Universal Robots PolyScope program: tarea_comandos.urp

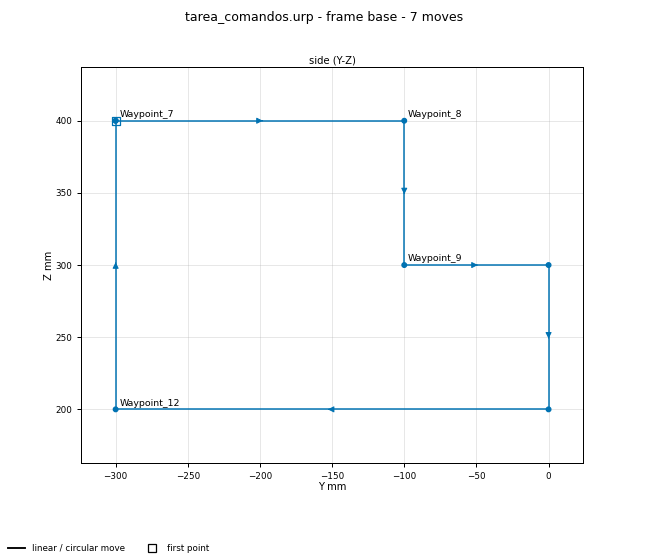
[picture p0: tool path of tarea_comandos.urp in frame base, 7 of 14 moves have a stored position in this frame; points joined in program order, loops and branches not executed]
Program tarea_comandos (installation=default directory=/home/hugo/Documents/Proyecto_Ingenieria/ursim-5.10.2.106319/programs/ASM/Clase1_Comandos createdIn=5.10.2.106319 lastSavedIn=5.10.2.106319 robotSerialNumber=20195599999)
Calibrated DH parameters: a=[0, -0.425, -0.3922, 0, 0, 0]; d=[0.1625, 0, 0, 0.1333, 0.0997, 0.0996]; alpha=[1.570796, 0, 0, 1.570796, -1.570796, 0]; deltaTheta=[0, 0, 0, 0, 0, 0]
Robot Program (runOnlyOnce=false)
  movimiento :=  (valueSource=Operator message=Elige Movimiento [1 - Relativos, 2 - Absolutos, 3 - Problema] valueType=Integer)
  repeticiones :=  (valueSource=Operator message=Introduce cantidad de repeticiones valueType=Integer)
  Loop While (checkContinuously=false) expression=repeticiones
    Switch expression=movimiento
      Case (caseValue=1)
        Folder Movimiento 1
          MoveL speed 250 mm/s, acceleration 1200 mm/s^2 (useActiveTCP=true) feature=Base
            Waypoint Waypoint_1 (Relative): relativeFromPosition TCP in base x=200 y=-300 z=400 mm, rx=-0.0013 ry=3.1193 rz=0.0359 rad; joints [-35.148, -69.126, -119.753, -80.848, 91.806, 54.808] deg; TCP in base x=200 y=-300 z=400 mm, rx=-0.0013 ry=3.1193 rz=0.0359 rad; joints [-35.148, -69.126, -119.753, -80.848, 91.806, 54.808] deg
            Waypoint Waypoint_2 (Relative): relativeFromPosition TCP in base x=200 y=-300 z=400 mm, rx=-0.0012 ry=3.1163 rz=0.0389 rad; joints [-35.205, -69.129, -119.772, -80.75, 91.997, 54.757] deg; TCP in base x=200 y=-100 z=400 mm, rx=-0.0012 ry=3.1163 rz=0.0389 rad; joints [9.378, -42.937, -130.525, -94.888, 91.177, 99.35] deg
            Waypoint Waypoint_3 (Relative): relativeFromPosition TCP in base x=200 y=-100 z=400 mm, rx=-0.0012 ry=3.1163 rz=0.0389 rad; joints [9.378, -42.937, -130.525, -94.888, 91.177, 99.35] deg; TCP in base x=200 y=-100 z=300 mm, rx=-0.0012 ry=3.1163 rz=0.0389 rad; joints [9.378, -43.258, -145.11, -79.982, 91.177, 99.35] deg
            Waypoint Waypoint_4 (Relative): relativeFromPosition TCP in base x=200 y=-100 z=300 mm, rx=-0.0012 ry=3.1163 rz=0.0389 rad; joints [9.378, -43.258, -145.11, -79.982, 91.177, 99.35] deg; TCP in base x=200 y=0 z=300 mm, rx=-0.0012 ry=3.1163 rz=0.0389 rad; joints [41.723, -35.535, -146.437, -86.004, 90.112, 131.68] deg
            Waypoint Waypoint_5 (Relative): relativeFromPosition TCP in base x=200 y=0 z=300 mm, rx=-0.0012 ry=3.1163 rz=0.0389 rad; joints [41.723, -35.535, -146.437, -86.004, 90.112, 131.68] deg; TCP in base x=200 y=0 z=200 mm, rx=-0.0012 ry=3.1163 rz=0.0389 rad; joints [41.723, -41.975, -160.626, -65.375, 90.112, 131.68] deg
            Waypoint Waypoint_6 (Relative): relativeFromPosition TCP in base x=200 y=0 z=200 mm, rx=-0.0012 ry=3.1163 rz=0.0389 rad; joints [41.723, -41.975, -160.626, -65.375, 90.112, 131.68] deg; TCP in base x=200 y=-300 z=200 mm, rx=-0.0012 ry=3.1163 rz=0.0389 rad; joints [-35.205, -85.851, -141.282, -42.519, 91.997, 54.757] deg
            Waypoint Waypoint_13 (Relative): relativeFromPosition TCP in base x=200 y=-300 z=200 mm, rx=-0.0012 ry=3.1163 rz=0.0389 rad; joints [-35.205, -85.851, -141.282, -42.519, 91.997, 54.757] deg; TCP in base x=200 y=-300 z=400 mm, rx=-0.0012 ry=3.1163 rz=0.0389 rad; joints [-35.205, -69.129, -119.772, -80.75, 91.997, 54.757] deg
      Case (caseValue=2)
        Folder Movimiento 2
          MoveL speed 250 mm/s, acceleration 1200 mm/s^2 (useActiveTCP=true) feature=Base
            Waypoint Waypoint_7: TCP in base x=200 y=-300 z=400 mm, rx=-0.0013 ry=3.1195 rz=0.0358 rad; joints [-35.145, -69.126, -119.751, -80.853, 91.797, 54.811] deg
            Waypoint Waypoint_8: motionParameters(blendRadius=0.05); TCP in base x=200 y=-100 z=400 mm, rx=-0.0013 ry=3.1195 rz=0.0358 rad; joints [9.426, -42.984, -130.463, -95.1, 91.091, 99.391] deg
            Waypoint Waypoint_9: motionParameters(blendRadius=0.05); TCP in base x=200 y=-100 z=300 mm, rx=-0.0013 ry=3.1195 rz=0.0358 rad; joints [9.426, -43.298, -145.05, -80.2, 91.091, 99.391] deg
            Waypoint Waypoint_10: motionParameters(blendRadius=0.05); TCP in base x=200 y=0 z=300 mm, rx=-0.0013 ry=3.1195 rz=0.0358 rad; joints [41.7, -35.632, -146.369, -86.188, 90.147, 131.654] deg
            Waypoint Waypoint_11: TCP in base x=200 y=0 z=200 mm, rx=-0.0013 ry=3.1195 rz=0.0358 rad; joints [41.7, -42.069, -160.553, -65.567, 90.147, 131.654] deg
            Waypoint Waypoint_12: motionParameters(blendRadius=0.05); TCP in base x=200 y=-300 z=200 mm, rx=-0.0013 ry=3.1195 rz=0.0358 rad; joints [-35.145, -85.828, -141.27, -42.633, 91.797, 54.811] deg
            Waypoint Waypoint_7: TCP in base x=200 y=-300 z=400 mm, rx=-0.0013 ry=3.1195 rz=0.0358 rad; joints [-35.145, -69.126, -119.751, -80.853, 91.797, 54.811] deg
      Case (caseValue=3)
        Halt
      Case (caseValue=2147483647)
        Wait Sleep waitTime=0.5
    repeticiones := repeticiones-1
